{attribute addProperty BoxType "AT2000-0233-0022"}
{attribute addProperty Id "ControlAT %Q*UINT1621Current_setpoint_value_ChAT %Q*ARRAY[0 ..13] OF INT224280"}
{attribute addProperty CRC "3277034191"}
{attribute addProperty SizeInBites "240"}
{attribute addProperty SizeInBytes "30"}
TYPE CC_Outputs_14_Ch_8D55E481 :
STRUCT
	{attribute addProperty Name "Control"}
	Control AT %Q* : UINT;
	{attribute addProperty Name "Current_setpoint_value_Ch"}
	Current_setpoint_value_Ch AT %Q* : ARRAY[0 ..13] OF INT;
END_STRUCT
END_TYPE

(* stored: Version 1.2.0.0, ProductVersion 3.1.4024.9
   DUT CC_Outputs_14_Ch_8D55E481: Id {087fdf88-badd-477f-8d41-0dc62cabd598} *)
